{attribute 'GeneratedUsingTerminal: AT2041-0250-0018'}
{attribute addProperty BoxType "AT2041-0250-0018"}
{attribute addProperty Description "AT2041-0250 Motor module with feed, +45°, 250mm, 50V"}
{attribute addProperty Physics "YKY"}
{attribute addProperty Id "CC_InputsAT %I*CC_Inputs_2C1C9EE032CC_OutputsAT %Q*CC_Outputs_69F9BE1432WcStateAT %I*WcState_9091E0EB2InfoDataAT %I*InfoData_BEF6B88E18"}
{attribute addProperty CRC "782682559"}
{attribute addProperty Size "84"}
TYPE AT2041_2EA6C9BF EXTENDS EtcSlaveBoxBase_77A0E4A7 :
STRUCT
	{attribute addProperty Name "CC_Inputs"}
	CC_Inputs : CC_Inputs_2C1C9EE0;
	{attribute addProperty Name "CC_Outputs"}
	CC_Outputs : CC_Outputs_69F9BE14;
	{attribute addProperty Name "WcState"}
	WcState : WcState_9091E0EB;
	{attribute addProperty Name "InfoData"}
	InfoData : InfoData_BEF6B88E;
END_STRUCT
END_TYPE

(* stored: Version 1.2.0.0, ProductVersion 3.1.4024.11
   DUT AT2041_2EA6C9BF: Id {3298ec04-9ebb-4784-bbd5-80080ec0a39f} *)
